TYPE "LubrValve_Par"
VERSION : 0.1
// Block: LubrValve_Par
   STRUCT
      SystemOn : Bool;
      EnableCheckFdbk : Bool;
      CycleFdbkCheckTime : Time;
      WorkTime : Time;
      ValveONTime : Time;
      ValveOFFTime : Time;
      ValvePumpSetPoint : Int;
      LubrReqSetPoint : LReal;
   END_STRUCT;

END_TYPE
